// LS Electric XG5000 project: 통신성공프레임
// PLC LSPLC

PROGRAM NewProgram (task: 스캔 프로그램)

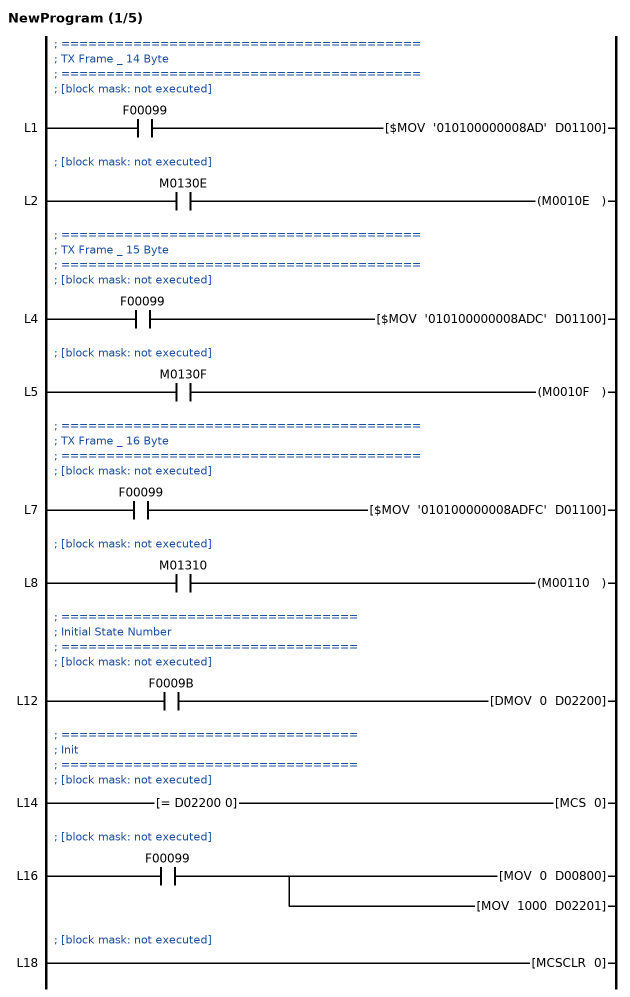
// ========================================
// TX Frame _ 14 Byte
// ========================================
; L1 (block mask: not executed)
LOAD      F00099
$MOV      '010100000008AD' D01100
; L2 (block mask: not executed)
LOAD      M0130E
OUT       M0010E
// ========================================
// TX Frame _ 15 Byte
// ========================================
; L4 (block mask: not executed)
LOAD      F00099
$MOV      '010100000008ADC' D01100
; L5 (block mask: not executed)
LOAD      M0130F
OUT       M0010F
// ========================================
// TX Frame _ 16 Byte
// ========================================
; L7 (block mask: not executed)
LOAD      F00099
$MOV      '010100000008ADFC' D01100
; L8 (block mask: not executed)
LOAD      M01310
OUT       M00110
// =================================
//    Initial State Number
// =================================
; L12 (block mask: not executed)
LOAD      F0009B
DMOV      0 D02200
// =================================
//    Init
// =================================
; L14 (block mask: not executed)
LOAD=     D02200 0
MCS       0
; L16 (block mask: not executed)
LOAD      F00099
MOV       0 D00800
MOV       1000 D02201
; L18 (block mask: not executed)
MCSCLR    0

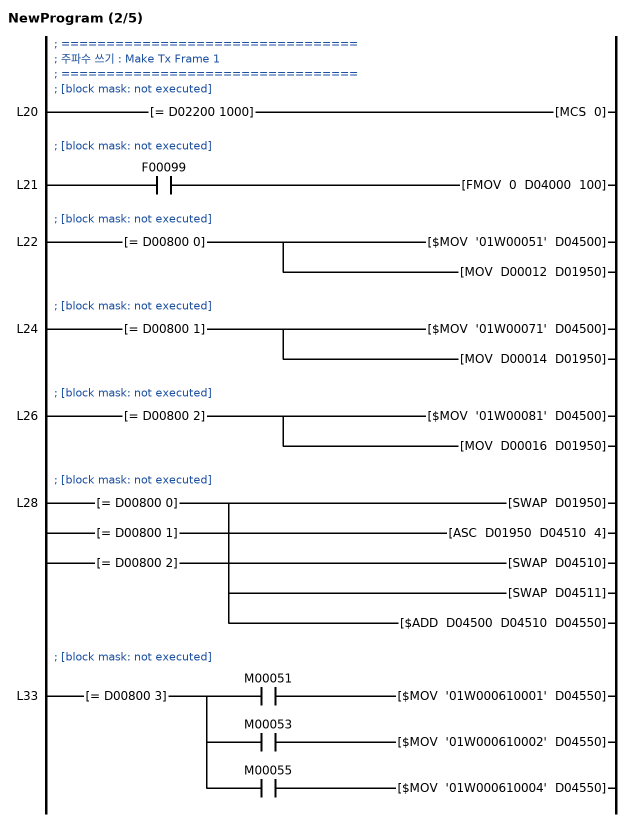
// =================================
//    주파수 쓰기 : Make Tx Frame 1
// =================================
; L20 (block mask: not executed)
LOAD=     D02200 1000
MCS       0
; L21 (block mask: not executed)
LOAD      F00099
FMOV      0 D04000 100
; L22 (block mask: not executed)
LOAD=     D00800 0
$MOV      '01W00051' D04500
MOV       D00012 D01950
; L24 (block mask: not executed)
LOAD=     D00800 1
$MOV      '01W00071' D04500
MOV       D00014 D01950
; L26 (block mask: not executed)
LOAD=     D00800 2
$MOV      '01W00081' D04500
MOV       D00016 D01950
; L28 (block mask: not executed)
LOAD=     D00800 0
OR=       D00800 1
OR=       D00800 2
SWAP      D01950
ASC       D01950 D04510 4
SWAP      D04510
SWAP      D04511
$ADD      D04500 D04510 D04550
; L33 (block mask: not executed)
LOAD=     D00800 3
MPUSH
AND       M00051
$MOV      '01W000610001' D04550
MLOAD
AND       M00053
$MOV      '01W000610002' D04550
MPOP
AND       M00055
$MOV      '01W000610004' D04550

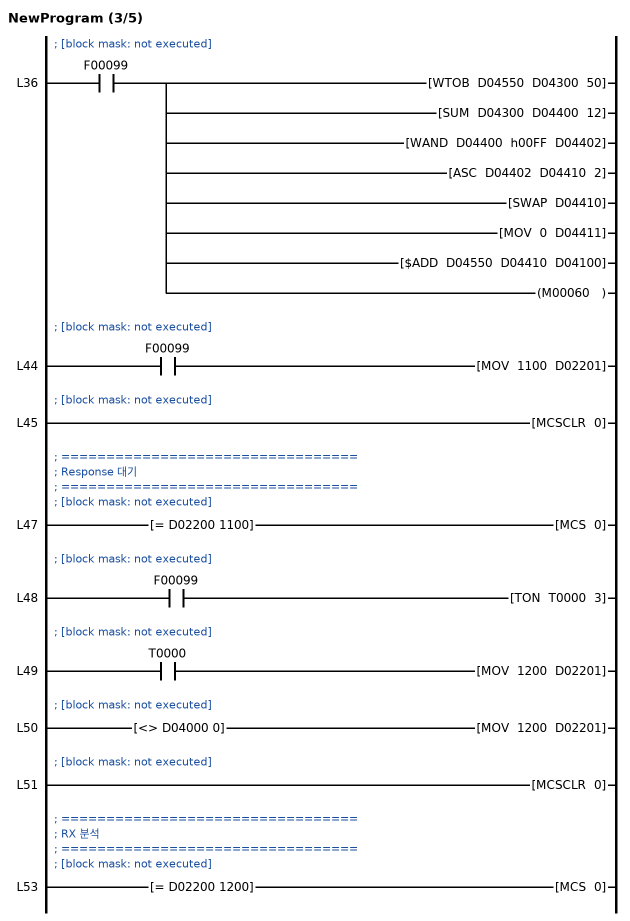
; L36 (block mask: not executed)
LOAD      F00099
WTOB      D04550 D04300 50
SUM       D04300 D04400 12
WAND      D04400 h00FF D04402
ASC       D04402 D04410 2
SWAP      D04410
MOV       0 D04411
$ADD      D04550 D04410 D04100
OUT       M00060
; L44 (block mask: not executed)
LOAD      F00099
MOV       1100 D02201
; L45 (block mask: not executed)
MCSCLR    0
// =================================
//    Response 대기
// =================================
; L47 (block mask: not executed)
LOAD=     D02200 1100
MCS       0
; L48 (block mask: not executed)
LOAD      F00099
TON       T0000 3
; L49 (block mask: not executed)
LOAD      T0000
MOV       1200 D02201
; L50 (block mask: not executed)
LOAD<>    D04000 0
MOV       1200 D02201
; L51 (block mask: not executed)
MCSCLR    0
// =================================
//    RX 분석
// =================================
; L53 (block mask: not executed)
LOAD=     D02200 1200
MCS       0

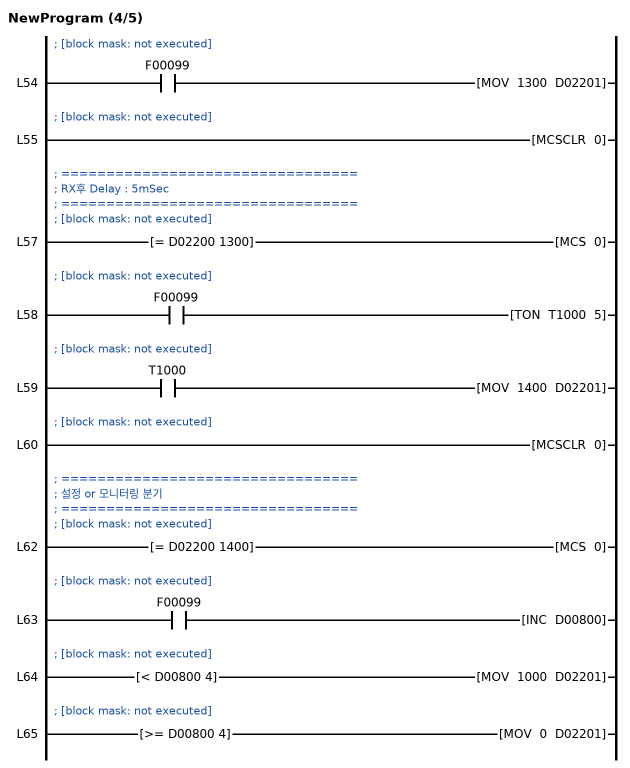
; L54 (block mask: not executed)
LOAD      F00099
MOV       1300 D02201
; L55 (block mask: not executed)
MCSCLR    0
// =================================
//    RX후 Delay : 5mSec
// =================================
; L57 (block mask: not executed)
LOAD=     D02200 1300
MCS       0
; L58 (block mask: not executed)
LOAD      F00099
TON       T1000 5
; L59 (block mask: not executed)
LOAD      T1000
MOV       1400 D02201
; L60 (block mask: not executed)
MCSCLR    0
// =================================
//    설정 or 모니터링 분기
// =================================
; L62 (block mask: not executed)
LOAD=     D02200 1400
MCS       0
; L63 (block mask: not executed)
LOAD      F00099
INC       D00800
; L64 (block mask: not executed)
LOAD<     D00800 4
MOV       1000 D02201
; L65 (block mask: not executed)
LOAD>=    D00800 4
MOV       0 D02201

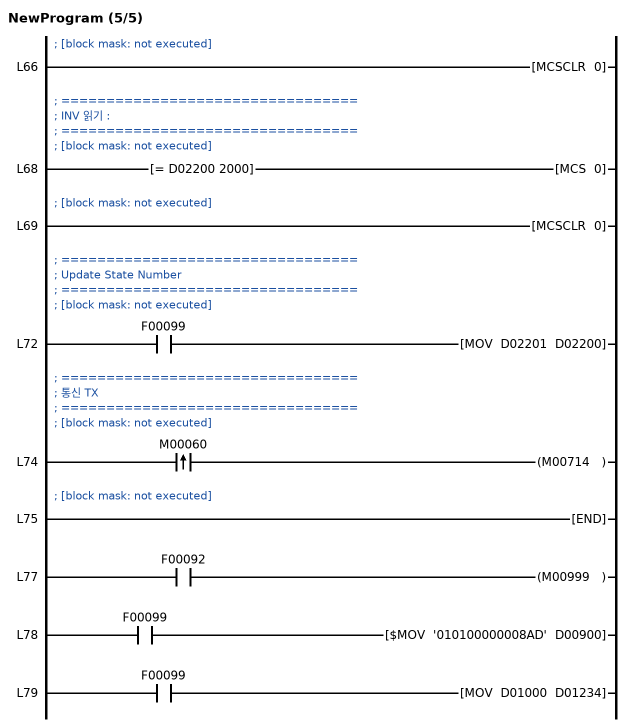
; L66 (block mask: not executed)
MCSCLR    0
// =================================
//    INV 읽기 :
// =================================
; L68 (block mask: not executed)
LOAD=     D02200 2000
MCS       0
; L69 (block mask: not executed)
MCSCLR    0
// =================================
//    Update State Number
// =================================
; L72 (block mask: not executed)
LOAD      F00099
MOV       D02201 D02200
// =================================
//    통신 TX
// =================================
; L74 (block mask: not executed)
LOADP     M00060
OUT       M00714
; L75 (block mask: not executed)
END
; L77
LOAD      F00092
OUT       M00999
; L78
LOAD      F00099
$MOV      '010100000008AD' D00900
; L79
LOAD      F00099
MOV       D01000 D01234